PROGRAM prgComLynus
VAR
	fbCom			: FB_MqttCommunicator_V2;
END_VAR

fbCom(
	bConnect:= TRUE, 
	strAuthKey:= 'TSG88376368072' , 
	sUserName:= 'a242cb33-7d00-431c-a780-261995d86f3c', 
	sUserPassword:= '68bc2b87-a9ad-4107-814c-33cbf7ba0678' , 
	eSavePositionCertificate:= eSavePositionOnPLC.ePostionHardDisk,  
	bConnected=> , 
	bError=> , 
	hrErrorCode=> , 
	eConnectionState=> , 
	eErrorMessage_Out=> );

(*
fbCom(
	bConnect:= TRUE, 
	sUserName:= 'a242cb33-7d00-431c-a780-261995d86f3c', 
	sUserPassword:= '68bc2b87-a9ad-4107-814c-33cbf7ba0678', 
	eSavePositionCertificate:= eSavePositionOnPLC.ePostionHardDisk, 
	bConnected=> , 
	bError=> , 
	hrErrorCode=> , 
	eConnectionState=> , 
	eErrorMessage_Out=> );
*)

END_PROGRAM

(* stored: Version 1.1.0.1, ProductVersion 3.1.4024.11
   POU prgComLynus: Id {64c3386a-a78c-459d-aa5f-2c9876969cae}, SpecialFunc None *)
